{attribute 'enable_dynamic_creation'}
FUNCTION_BLOCK FB_Red IMPLEMENTS I_Color
VAR_INPUT
END_VAR
VAR_OUTPUT
END_VAR
VAR
END_VAR


METHOD M_Fill : BOOL
ADSLOGSTR(ADSLOG_MSGTYPE_HINT, 'Paint Red', '');
M_Fill := TRUE;
END_METHOD

END_FUNCTION_BLOCK

(* stored: Version 1.1.0.1, ProductVersion 3.1.4024.12
   POU FB_Red: Id {3af52522-8a45-41d6-940a-4988b9b31cf6}, SpecialFunc None
   Method M_Fill: Id {69db6a5a-b341-4515-9fd5-68d949a4e314} *)
